// TIA Portal V19 export
TYPE "typeAxisControlInterface"
// stored: Access Published
   STRUCT
      manual : "typeAxisControlManual";
      production : "typeAxisControlProduction";
      maintenance { S7_SetPoint := 'True'} : "typeAxisControlMaintenance";
   END_STRUCT;
END_TYPE
